// Brief: Slave Arm Adjust
FUNCTION_BLOCK PUBLIC FB_SlaveCtrlDargFreeTest EXTENDS FB_SlaveArmCtrlBase
VAR
	// velocity for full damping
	m_maxAdjustVel :Vec3d := [1.2, 1.2, 0.3];
	
	// velocity start to enable damping
	m_velLBForDamp :Vec3d := [0.7, 0.7, 0.1];
	
	// max damp
	m_maxDamp :Vec3d := [1,1,100];//50, 50, 500
	
	// distance buffer from joint limit to start damp
	m_limitBufferForDamp :Vec3d :=[20*g_deg2Rad, 20*g_deg2Rad, 0.03];
	
	//joint limit position
	m_DHjntPos:Vec8d;
	m_jntPosMin:Vec8d;
	m_jntPosMax:Vec8d;
	m_jntMotRange:Vec8d;
	
	//unit transform
	m_unitTransform:FB_UnitTransform;
END_VAR

// override this function in each exact controller
METHOD PROTECTED calcCmdJntPos : BOOL
VAR_IN_OUT CONSTANT
	i_endoscopePose : ST_Frame;
	i_masterStatus :ST_MasterStatus;
	i_setupStatus: ST_SetupStatus;
	i_slaveArm :FB_SlaveArm;
END_VAR
VAR
	i:INT;
END_VAR

(*
m_cmdJntPos[1]:=i_slaveArm.curJntPos[1];
m_cmdJntPos[2]:=i_slaveArm.curJntPos[2];
m_cmdJntPos[3]:=i_slaveArm.curJntPos[3];
FOR i:= 6 TO 8 DO
	IF m_jntOPMode[i] = DriverOPMode_Trq THEN
		m_cmdJntPos[i]:=i_slaveArm.curJntPos[i];
	END_IF
END_FOR

m_cmdCartPose:=i_slaveArm.curCartPose;
*)

//add code for test
FOR i:=1 TO 8 BY 1 DO
	IF (g_motionRangeTest.m_slaveJntEnable[i]=TRUE) THEN
		m_jntEnableFlag[i]:=1;
	ELSE
		m_jntEnableFlag[i]:=0;
	END_IF
END_FOR

//copy the current joint position to command joint position
m_cmdJntPos:=i_slaveArm.curJntPos;
m_cmdCartPose:=i_slaveArm.curCartPose;

//Calculate the LIMIT value
m_DHjntPos:=i_slaveArm.curJntPos;
FOR i:=1 TO 8 BY 1 DO
	IF (m_DHjntPos[i]>m_jntPosMax[i]) THEN
		m_jntPosMax[i]:=m_DHjntPos[i];
	ELSIF (m_DHjntPos[i]<m_jntPosMin[i]) THEN
		m_jntPosMin[i]:=m_DHjntPos[i];
	END_IF
END_FOR
vecSub(m_jntPosMax,m_jntPosMin,m_jntMotRange);

//feedback the information
i:=i_slaveArm.armIdx;
g_motionRangeTest.m_slaveJntPos[i]:=m_unitTransform.slaveArmUnit2UserN8(m_DHjntPos);
g_motionRangeTest.m_slaveJntPosMin[i]:=m_unitTransform.slaveArmUnit2UserN8(m_jntPosMin);
g_motionRangeTest.m_slaveJntPosMax[i]:=m_unitTransform.slaveArmUnit2UserN8(m_jntPosMax);
g_motionRangeTest.m_slaveJntPosRange[i]:=m_unitTransform.slaveArmUnit2UserN8(m_jntMotRange);
END_METHOD

// override this function in each exact controller
METHOD PROTECTED calcCmdJntTrq : BOOL
VAR_IN_OUT CONSTANT
	i_endoscopePose : ST_Frame;
	i_masterStatus :ST_MasterStatus;
	i_setupStatus: ST_SetupStatus;
	i_slaveArm :FB_SlaveArm;
END_VAR
VAR
	i :INT;
	dampScale :LREAL;
	limitDis:LREAL;
END_VAR
(*
// set joint torque to zero in default
m_cmdJntTrq := g_zeroVec8d;

// enable endoscope rotation joint if external torque exceed specific value
IF i_slaveArm.instrument.onChipData.m_InstruReadSucceed AND i_slaveArm.instrument.instruType = InstruType_Endoscope THEN
		FOR i:=6 TO 8 DO 
			IF ABS(i_slaveArm.filtJntCurrent[i]) > 100 THEN
				m_jntOPMode[i]:=DriverOPMode_Trq;
			END_IF
		END_FOR
END_IF

// add damp near joint limit
FOR i:=1 TO 3 DO
	IF (i_slaveArm.curJntPos[i] > GVL_SlaveMotorParameters.g_maxDHJntPos[i] - m_limitBufferForDamp[i] AND  i_slaveArm.curJntVel[i]> 0 ) 
		OR (i_slaveArm.curJntPos[i] < GVL_SlaveMotorParameters.g_minDHJntPos[i] + m_limitBufferForDamp[i] AND  i_slaveArm.curJntVel[i]<0 )  THEN
		limitDis := MIN(GVL_SlaveMotorParameters.g_maxDHJntPos[i] - i_slaveArm.curJntPos[i], i_slaveArm.curJntPos[i]-GVL_SlaveMotorParameters.g_minDHJntPos[i]);
		dampScale  :=LIMIT(0, 1-limitDis/m_limitBufferForDamp[i],1);
		m_cmdJntTrq[i]:= -dampScale * m_maxDamp[i] * i_slaveArm.curJntVel[i];
	END_IF
	
END_FOR

// compute damp
FOR i:=1 TO 3 DO
	IF ABS(i_slaveArm.curJntVel[i]) > m_velLBForDamp[i] THEN 
		dampScale:=LIMIT(0, (ABS(i_slaveArm.curJntVel[i])- m_velLBForDamp[i])/(m_maxAdjustVel[i] - m_velLBForDamp[i]), 1 );
		m_cmdJntTrq[i] :=m_cmdJntTrq[i] -i_slaveArm.curJntVel[i] * m_maxDamp[i] * dampScale;
	END_IF
END_FOR
*)

m_cmdJntTrq := g_zeroVec8d;
END_METHOD

METHOD PUBLIC init : BOOL
VAR_IN_OUT CONSTANT
	i_slaveArm	:FB_SlaveArm;
END_VAR
VAR_IN_OUT 
	r_slaveArmCtrlCmd :ST_SlaveArmCtrlCmds;
END_VAR
VAR
	i :INT;
END_VAR
// check if to hold the command joint position unchanged
m_holdLastCmds := checkToHoldLastCmds(i_slaveArm);

//init
SUPER^.Init(i_slaveArm,r_slaveArmCtrlCmd);

// disable joints if this joint is an unrecoverable failure
FOR i:=1 TO g_sJntNum DO
	IF SafetyCheck.m_SafetyCheck.m_jntErrFlag[i_slaveArm.armIdx, 0, 3] OR  SafetyCheck.m_SafetyCheck.m_jntErrFlag[i_slaveArm.armIdx, i+g_setupJntNum, 3] THEN
		m_jntEnableFlag[i] := 0;
	ELSE
		m_jntEnableFlag[i] := 1;
	END_IF
END_FOR

// joint 1/2/3/7 run in torque mode
m_jntOPMode[1]:=DriverOPMode_Trq;
m_jntOPMode[2]:=DriverOPMode_Trq;
m_jntOPMode[3]:=DriverOPMode_Trq;
m_jntOPMode[4]:=DriverOPMode_PosTrq;
m_jntOPMode[5]:=DriverOPMode_PosTrq;
m_jntOPMode[6]:=DriverOPMode_PosTrq;
m_jntOPMode[7]:=DriverOPMode_PosTrq;
m_jntOPMode[8]:=DriverOPMode_PosTrq;

IF i_slaveArm.instrument.onChipData.m_InstruReadSucceed THEN
	IF i_slaveArm.instrument.instruType <> InstruType_Endoscope THEN
		m_jntOPMode[7]:=DriverOPMode_Trq;
	END_IF
END_IF

// update commands to arm
copyCmds(r_slaveArmCtrlCmd);


//add code for test
FOR i:=1 TO 8 BY 1 DO
	IF (g_motionRangeTest.m_slaveJntEnable[i]=TRUE) THEN
		m_jntEnableFlag[i]:=1;
	ELSE
		m_jntEnableFlag[i]:=0;
	END_IF
END_FOR

m_jntOPMode:=g_slaveAllTrqMode;
m_DHjntPos:=i_slaveArm.curJntPos;
m_jntPosMin:=m_DHjntPos;
m_jntPosMax:=m_DHjntPos;
vecSub(m_jntPosMax,m_jntPosMin,m_jntMotRange);
END_METHOD

END_FUNCTION_BLOCK

(* stored: Version 1.1.0.1, ProductVersion 3.1.4024.11
   POU FB_SlaveCtrlDargFreeTest: Id {56556deb-8915-4729-97e3-a8f7e4569550}, SpecialFunc None
   Method calcCmdJntPos: Id {5cedd5a0-fa85-48d9-a6b4-18b50cbe2fb3}
   Method calcCmdJntTrq: Id {b3fabaf1-5d32-4e53-9850-80423e860bf4}
   Method init: Id {43ae67a2-b72a-4026-9dbb-dae4546670be} *)
